(* PLC project Unnamed, Unknown Unnamed 1 *)
(* stored: creationDateTime 2025-10-12T20:06:37, modificationDateTime 2025-10-13T07:20:51 *)

PROGRAM Main_Program
  VAR_INPUT
    myPI : PID;
  END_VAR
  VAR_EXTERNAL
    CV : REAL;
    SP : REAL;
    PV : REAL;
  END_VAR
  VAR
    error : REAL;
    Ki : REAL;
    Kp : REAL;
    I_accumulator : REAL;
    Ts : REAL;
    I_accumulator1 : REAL;
  END_VAR

            Kp := 50.0;

Ki := 0.0001;

Ts := 0.02;



error := SP - PV;

I_accumulator := I_accumulator + Ki * error * Ts;

CV := Kp * error + I_accumulator;
          
END_PROGRAM

CONFIGURATION Config0
  RESOURCE Res0 ON PLC
    VAR_GLOBAL
      CV : REAL;
      PV : REAL;
      SP : REAL;
    END_VAR
    TASK task0(INTERVAL := T#20ms, PRIORITY := 0);
    PROGRAM instance0 WITH task0 : Main_Program;
  END_RESOURCE
END_CONFIGURATION
